TYPE ST_GripperCommunicationConfig :
STRUCT
    tAdsTimeout : TIME;
    tPollInterval : TIME;
END_STRUCT
END_TYPE

(* stored: Version 1.1.0.1, ProductVersion 3.1.4026.20
   DUT ST_GripperCommunicationConfig: Id {e9dcd49c-4b6d-4b9e-bd52-32b948444673} *)
